(* CoDeSys 2.3.9.415 project: exercise_6.pro *)
(* Libraries: STANDARD.LIB 4.10.05 11:14:46, IECSFC.LIB 13.4.06 15:51:28, ANALYZATION.LIB 5.10.99 09:05:06, SysLibCom.lib 19.1.24 11:13:16, ComService.lib 21.5.09 13:28:28, ModBus.lib 19.1.24 10:36:34, Util.lib 18.5.10 15:14:28 *)

(* PLC configuration (modules and I/O channels)
PLC100.K [Root] node -1, in %IB0 out %QB0 {MinCycleLength = 1; MaxCycleLength = 1000}
  Discrete input 8 bit [ID100] node 0, in %IB0 out %QB0 {Filtrationtime = 10; Filtrationtime = 10; Filtrationtime = 10; Filtrationtime = 10; Filtrationtime = 10; Filtrationtime = 10; Filtrationtime = 10; Filtrationtime = 10; Visibility = No; PinCount = 8; WatchDogPeriod = 1000; PollPeriod = 1}
    AT %IB0.0 [ByteInput] 8 discrete inputs
  Discrete output 2 bit [ID101] node 1, in %IB1 out %QB1 {PinCount = 2; SafeValueBool = FALSE; SafeValueBool = FALSE; Visibility = No}
    AT %QX1.0 [BitOutput] First
    AT %QX1.1 [BitOutput] Second
  Discrete output 2 bit [ID101] node 2, in %IB2 out %QB2 {PinCount = 2; SafeValueBool = FALSE; SafeValueBool = FALSE; Visibility = No}
    AT %QX2.0 [BitOutput] First
    AT %QX2.1 [BitOutput] Second
  Discrete output 2 bit [ID101] node 3, in %IB3 out %QB3 {PinCount = 2; SafeValueBool = FALSE; SafeValueBool = FALSE; Visibility = No}
    AT %QX3.0 [BitOutput] First
    AT %QX3.1 [BitOutput] Second
  Discrete output 2 bit [ID101] node 4, in %IB4 out %QB4 {PinCount = 2; SafeValueBool = FALSE; SafeValueBool = FALSE; Visibility = No}
    AT %QX4.0 [BitOutput] First
    AT %QX4.1 [BitOutput] Second
  Discrete output 2 bit [ID101] node 5, in %IB5 out %QB5 {PinCount = 2; SafeValueBool = FALSE; SafeValueBool = FALSE; Visibility = No}
    AT %QX5.0 [BitOutput] First
    AT %QX5.1 [BitOutput] Second
  Discrete output 2 bit [ID101] node 6, in %IB6 out %QB6 {PinCount = 2; SafeValueBool = FALSE; SafeValueBool = FALSE; Visibility = No}
    AT %QX6.0 [BitOutput] First
    AT %QX6.1 [BitOutput] Second
  Special output [ID104] node 7, in %IB7 out %QB7 {Visibility = No; PinCount = 1}
    AT %QX7.0 [BitOutput] Special output
*)

(* Global variable list: Global_Variables *)
VAR_GLOBAL
	port_opened: BYTE := 0;
	Settings:COMSETTINGS;
	com_num: PORTS:=0;
	COM_SERVICE1: COM_SERVICE;

	Buffer: ARRAY[0..255] OF BYTE;
	Cmpl: ARRAY[0..30] OF BOOL;
	Err: ARRAY[0..30] OF BYTE;

	ModBusReadHoldReg:ARRAY [0..10] OF MB_RD_HOLD_REGS; (* FC3*)
	ModBusWriteMultiReg: ARRAY[0..10] OF MB_WR_REGS;
	ModBusSingleCoil: ARRAY[0..10] OF MB_WR_SNG_COIL; (*FC5*)

	NumberSend: BYTE;

	In: WORD;
	Out: WORD;

	TonConnect: ARRAY[0..3] OF TON;
	ToffConnect: ARRAY[0..3] OF TOF;
	ConnectionStatus: ARRAY [0..3] OF BOOL;

	DiodStats: BOOL;

	timer1: TON;
	i: BYTE;

	stop: BOOL;

	Timer: TON;
	Triger: R_TRIG;

	(*Новые переменые*)

	SwitchDisplayStat: BOOL;
	password: BYTE;

	test: WORD := 2#0000_0000_0000_0001;
	aaa: F_TRIG;
	i1: BYTE;
	variableTemp: WORD;

END_VAR
VAR_GLOBAL RETAIN
  Variable: WORD := 5;
END_VAR

(* POU PLC_PRG, ST *)
PROGRAM PLC_PRG
VAR
	start: BOOL;
END_VAR
IF start=0 THEN
	Init();
	start:=1;
	in.15 := TRUE;
END_IF
Link();

ButtonOn();
RunLight();
SwitchDisplay();
ChangeMenu();

IF IN.15 = FALSE THEN
	stop := TRUE;
	DiodStats := FALSE;
END_IF

IF  stop THEN
	RETURN;
END_IF
END_PROGRAM

(* POU Init, ST *)
FUNCTION Init : BOOL
VAR_INPUT
END_VAR
VAR
END_VAR
WHILE port_opened=0 DO
	IF port_opened=0 THEN
		Settings.Port:=com_num;
		Settings.dwBaudRate:=57600;
		Settings.byParity:=0;
		Settings.dwTimeout:=0;
		Settings.byStopBits:=0;
		Settings.dwBufferSize:=0;
		Settings.dwScan:=0;
	END_IF

	COM_SERVICE1(Enable:=(port_opened=0), Settings:=Settings, Task:= OPEN_TSK );

	IF COM_SERVICE1.ready THEN
		port_opened:=2;
	END_IF
END_WHILE
END_FUNCTION

(* POU Link, ST *)
FUNCTION Link : BOOL
VAR
	z: BYTE;
	a: BOOL;
END_VAR
CASE NumberSend OF
0:
            Buffer[1]:=WORD_TO_BYTE(Out AND 16#00FF);
		Buffer[0]:=WORD_TO_BYTE(SHR(Out, 8));

	       ModBusWriteMultiReg[0](
			Enable:=TRUE ,
			Mode:=MB_RTU ,
			DevAddr:=4, (* адрес *)
			FirstAddr:=0 ,
			Quantity:=1 ,
			ComHandle:=Settings.Port ,
			TimeOut:=T#50ms ,
			Buffer:=Buffer,
	       	Complete=>Cmpl[0] ,
			Exception=>Err[0] ,
			RegCnt=>
		);

		IF(cmpl[0]=TRUE) THEN
			NumberSend:=1;
		END_IF
1:
	ModBusReadHoldReg[0](
		Enable:=TRUE ,
		Mode:=MB_RTU ,
		DevAddr:=4, (* адрес *)
		FirstAddr:=1 ,
		Quantity:=1 ,
		ComHandle:=Settings.Port,
		TimeOut:=T#50ms,
		Buffer:=Buffer,
		Complete=>Cmpl[1],
		Exception=>Err[1] ,
		ByteCnt=>
	 );

	      IF(cmpl[1]=TRUE) THEN
			IF (Err[1]=0) THEN
				In:=SHL(Buffer[0], 8)+Buffer[1];
			END_IF
			TonConnect[0](IN:=((Err[1])<>0) , PT:=T#5s  , Q=>a , ET=> );
			ToffConnect[0](IN:=a , PT:=T#10s , Q=>ConnectionStatus[0] , ET=> );
			NumberSend:=2;
		END_IF
2:
	Buffer[1]:=WORD_TO_BYTE(Out AND 16#00FF);
	Buffer[0]:=WORD_TO_BYTE(SHR(Out, 8));

	ModBusWriteMultiReg[1](
		Enable:=TRUE ,
		Mode:=MB_RTU ,
		DevAddr:=6, (* адрес *)
		FirstAddr:=300 ,
		Quantity:=1,
		ComHandle:=Settings.Port ,
		TimeOut:=T#50ms ,
		Buffer:=Buffer,
	       Complete=>Cmpl[2] ,
		Exception=>Err[2] ,
		RegCnt=>
	);

	IF(cmpl[2]=TRUE) THEN
		NumberSend:=3;
	END_IF
3:
	ModBusSingleCoil[0](
		Enable := TRUE,
		Mode := MB_RTU,
		DevAddr := 6, (* адрес *)
		CoilAddr := 272,
		Value := in.0 OR DiodStats,
		ComHandle := Settings.Port,
		TimeOut := T#50ms,

		Complete => Cmpl[3],
		Exception => Err[3],
	);

	IF(cmpl[3]=TRUE) THEN
			NumberSend:=4;
	END_IF
4:
	ModBusSingleCoil[1](
		Enable := TRUE,
		Mode := MB_RTU,
		DevAddr := 6, (* адрес *)
		CoilAddr := 273,
		Value := NOT in.15,
		ComHandle := Settings.Port,
		TimeOut := T#50ms,

		Complete => Cmpl[4],
		Exception => Err[4],
	);


	IF(cmpl[4]=TRUE) THEN
			NumberSend:=5;
	END_IF
5: (*Переключение экранов*)
	Buffer[1]:=WORD_TO_BYTE(In AND 16#00FF);
	Buffer[0]:=WORD_TO_BYTE(SHR(in, 7));

	ModBusSingleCoil[2](
		Enable := TRUE,
		Mode := MB_RTU,
		DevAddr := 6, (* адрес *)
		CoilAddr := 256,
		Value := SwitchDisplayStat,
		ComHandle := Settings.Port,
		TimeOut := T#50ms,

	       Complete=>Cmpl[5] ,
		Exception=>Err[5] ,
	);
	IF(cmpl[5]=TRUE) THEN
			NumberSend:=6;
	END_IF
6: (*Пароль*)
	ModBusReadHoldReg[1](
		Enable:=TRUE ,
		Mode:=MB_RTU ,
		DevAddr:=6, (* адрес *)
		FirstAddr:=347 ,
		Quantity:=4,
		ComHandle:=Settings.Port,
		TimeOut:=T#50ms,
		Buffer:=Buffer,
		Complete=>Cmpl[6],
		Exception=>Err[6],
		ByteCnt=>
	 );

	IF(cmpl[6]=TRUE) THEN
			IF (Err[6]=0) THEN
				password := SHL(Buffer[0], 8)+Buffer[1];
			END_IF
			TonConnect[1](IN:=((Err[1])<>0) , PT:=T#5s  , Q=>a , ET=> );
			ToffConnect[1](IN:=a , PT:=T#10s , Q=>ConnectionStatus[1] , ET=> );
			NumberSend:=7;
	END_IF
7:
	Buffer[1]:=WORD_TO_BYTE(test AND 16#00FF);
	Buffer[0]:=WORD_TO_BYTE(SHR(test, 8));

	ModBusWriteMultiReg[2](
		Enable:=TRUE ,
		Mode:=MB_RTU ,
		DevAddr:=6, (* адрес *)
		FirstAddr:=351,
		Quantity:=1,
		ComHandle:=Settings.Port ,
		TimeOut:=T#50ms ,
		Buffer:=Buffer,
	       Complete=>Cmpl[7] ,
		Exception=>Err[7],
		RegCnt=>
	);

	IF(cmpl[7]=TRUE) THEN
		NumberSend:=8;
	END_IF
8:
	Buffer[1]:=WORD_TO_BYTE(Variable AND 16#00FF);
	Buffer[0]:=WORD_TO_BYTE(SHR(Variable, 8));

	ModBusWriteMultiReg[3](
		Enable:=TRUE ,
		Mode:=MB_RTU ,
		DevAddr:=6, (* адрес *)
		FirstAddr:=352,
		Quantity:=1,
		ComHandle:=Settings.Port ,
		TimeOut:=T#50ms ,
		Buffer:=Buffer,
	       Complete=>Cmpl[8] ,
		Exception=>Err[8],
		RegCnt=>
	);

	IF(cmpl[8]=TRUE) THEN
		NumberSend:=0;
	END_IF
END_CASE
END_FUNCTION

(* POU ButtonOn, ST *)
FUNCTION ButtonOn : BOOL
VAR_INPUT
END_VAR
VAR
END_VAR
Timer(
	IN := in.0,
	PT := T#1s,
);

Triger( CLK := 	Timer.Q );

DiodStats := Triger.Q XOR DiodStats;

IF Triger.Q = TRUE THEN
	stop := FALSE;
END_IF
END_FUNCTION

(* POU RunLight, ST *)
FUNCTION RunLight : BOOL
VAR_INPUT
END_VAR
VAR
END_VAR
IF DiodStats = TRUE THEN
	timer1(IN := NOT timer1.Q, PT := t#500MS);

	IF timer1.Q THEN

		IF i = 0 THEN
			OUT := 16#1;
		ELSE
			OUT :=  SHL(WORD#1,  i);
		END_IF

		i := i + 2;
	END_IF

ELSE
	OUT := i := 0;
END_IF

IF i >= 16 THEN
	i := 0;
END_IF
END_FUNCTION

(* POU SwitchDisplay, ST *)
FUNCTION SwitchDisplay : BOOL
VAR_INPUT
END_VAR
VAR
END_VAR
SwitchDisplayStat := in.4;
END_FUNCTION

(* POU ChangeMenu, ST *)
FUNCTION ChangeMenu : BOOL
VAR_INPUT
END_VAR
VAR
END_VAR
(*aaa(CLK := in.2);

in.2;
aaa.Q;*)

aaa(CLK := in.2);

IF aaa.Q THEN
	i1 := i1 + 1;
	test := SHL( test, 1 );
END_IF

IF i1 >= 3 THEN
	i1 := 1;
	test := 1;
END_IF
END_FUNCTION
